TYPE MachineOperationMode :
STRUCT
	AUTO	: BOOL;
	MANUAL	: BOOL;
END_STRUCT
END_TYPE

(* stored: Version 1.1.0.1, ProductVersion 3.1.4024.11
   DUT MachineOperationMode: Id {37257248-6923-435a-9937-e8c737d6dbb8} *)
